FUNCTION_BLOCK FB_MotionLogger IMPLEMENTS I_MotionLogger
VAR_INPUT
END_VAR
VAR_OUTPUT
END_VAR
VAR
END_VAR

END_FUNCTION_BLOCK

(* stored: Version 1.1.0.1
   POU FB_MotionLogger: Id {6fbb242a-2ddb-457e-b22a-4be4b700b56a}, SpecialFunc None *)
